Omron Sysmac Studio project CC087 Control System Demo 2.0 (Sysmac Studio 1.0.8.31, StandardProject)

# Controller new_Controller_0: NJ301-1100 version 1.6
Axis MC_Axis000, settings changed from default: AxisType=ServoType, HomingMode=LimitSignalOff, OriginInputMode=EXT, HomingVelocity=100000, HomingApproachVelocity=10000, OriginPositionOffset=1000
Task PrimaryTask (priority 4, period or condition 1000): Program0

VAR_GLOBAL
    CounterVariable1 : INT := 0;
    NB_Size AT %W3 : INT := 0;
    NB_Color AT %W4 : INT;
END_VAR
VAR_GLOBAL RETAIN
    ErrorMessage AT %H0.02 : BOOL;
END_VAR
VAR_GLOBAL
    NumberSelected : INT := 0;
    NB_A AT %W0.08 : BOOL;
    NB_B AT %W0.10 : BOOL;
    NB_C AT %W0.11 : BOOL;
    NB_D AT %W0.12 : BOOL;
    NB_E AT %W0.13 : BOOL;
    NB_F AT %W0.14 : BOOL;
    NB_G AT %W0.15 : BOOL;
END_VAR
VAR_GLOBAL RETAIN
    NB_Black AT %H0.01 : BOOL;
END_VAR
VAR_GLOBAL
    NB_Blue AT %W0.09 : BOOL;
    NB_Green AT %W0.07 : BOOL;
    NB_OutputWord AT %W2 : STRING[256];
    NB_Word AT %W1 : INT;
    NB_Run AT %W0.02 : BOOL;
    NB_Power AT %W0.03 : BOOL;
    CounterVariable2 : INT := 0;
    CounterVariable3 : INT := 0;
    Motor : BOOL;
    GreenStartButtonLight : BOOL;  (* at ECAT://node#[2,2]/Output Bit 16 bits/Output Bit 03 *)
    SwOne : BOOL;
    SwTwo : BOOL;
    SwThree : BOOL;
    SwFour : BOOL;
    OutOne : BOOL;  (* at ECAT://node#[2,2]/Output Bit 16 bits/Output Bit 04 *)
    OutTwo : BOOL;  (* at ECAT://node#[2,2]/Output Bit 16 bits/Output Bit 05 *)
    OutThree : BOOL;  (* at ECAT://node#[2,2]/Output Bit 16 bits/Output Bit 06 *)
    OutFour : BOOL;  (* at ECAT://node#[2,2]/Output Bit 16 bits/Output Bit 07 *)
    OutFive : BOOL;
    ReadyStatus : BOOL;  (* at ECAT://node#[2,1]/Input Bit 16 bits/Input Bit 01 *)
    FaultStatus : BOOL;  (* at ECAT://node#[2,1]/Input Bit 16 bits/Input Bit 02 *)
    RunStatus : BOOL;
    ConditionOne : BOOL;  (* at ECAT://node#[2,1]/Input Bit 16 bits/Input Bit 00 *)
    ConditionTwo : BOOL;  (* at ECAT://node#[2,1]/Input Bit 16 bits/Input Bit 03 *)
    ConditionThree : BOOL;
    ConditionFour : BOOL;
    ConditionFive : BOOL;
    StandByMode : BOOL;
    GreenStackLight : BOOL;  (* at ECAT://node#[2,2]/Output Bit 16 bits/Output Bit 00 *)
    RedStackLight : BOOL;  (* at ECAT://node#[2,2]/Output Bit 16 bits/Output Bit 02 *)
    YellowStackLight : BOOL;  (* at ECAT://node#[2,2]/Output Bit 16 bits/Output Bit 01 *)
    Output1 : BOOL;
END_VAR
VAR_GLOBAL CONSTANT
    MC_Axis000 : _sAXIS_REF;  (* at MC://_MC_AX[0] *)
END_VAR

PROGRAM Program0
VAR
    DelayTimer1 : TON;
    ET1 : TIME;
    OnTimer1 : TP;
    ET2 : TIME;
    DelayTimer2 : TON;
    OnTimer2 : TP;
    ET3 : TIME;
    ET4 : TIME;
    DelayTimer3 : TON;
    OnTimer3 : TP;
    ET5 : TIME;
    ET6 : TIME;
    Output1 : BOOL;
    ConditionFour : BOOL;
    ConditionFive : BOOL;
    OutFive : BOOL;
    FaultTimer : TON;
    ET7 : TIME;
    Power1 : MC_Power;
    Move1 : MC_MoveRelative;
    Reset1 : MC_Reset;
    TestFunction : FunctionBlock0;
    TestInput : BOOL;
    TestOutput : BOOL;
    Output : BOOL;
    Fault : BOOL;
    Home1 : MC_Home;
END_VAR
VAR_EXTERNAL
    FaultStatus : BOOL;
    RedStackLight : BOOL;
    ReadyStatus : BOOL;
    YellowStackLight : BOOL;
    GreenStackLight : BOOL;
    StandByMode : BOOL;
    SwFour : BOOL;
    SwOne : BOOL;
    SwTwo : BOOL;
    SwThree : BOOL;
    GreenStartButtonLight : BOOL;
    ConditionOne : BOOL;
    ConditionTwo : BOOL;
    ConditionThree : BOOL;
    CounterVariable1 : INT;
    CounterVariable2 : INT;
    CounterVariable3 : INT;
    OutOne : BOOL;
    OutTwo : BOOL;
    OutThree : BOOL;
    OutFour : BOOL;
    NB_Run : BOOL;
END_VAR
VAR_EXTERNAL CONSTANT
    MC_Axis000 : _sAXIS_REF;
END_VAR
VAR_EXTERNAL
    NB_Power : BOOL;
    Motor : BOOL;
    NB_A : BOOL;
    NB_Green : BOOL;
    NB_OutputWord : STRING[256];
    NB_B : BOOL;
    NB_C : BOOL;
    NB_D : BOOL;
    NB_E : BOOL;
    NB_F : BOOL;
    NB_G : BOOL;
    NB_Black : BOOL;
    NB_Blue : BOOL;
    NumberSelected : INT;
    ErrorMessage : BOOL;
    NB_Size : INT;
    NB_Word : INT;
    NB_Color : INT;
END_VAR

(* Section Section0: ladder, written here as Structured Text *)

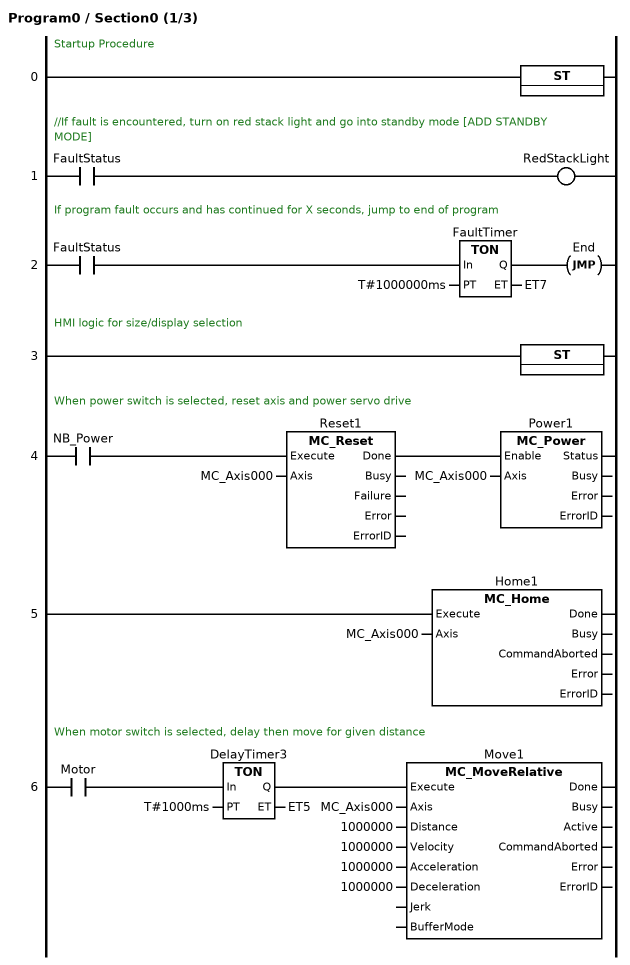
(* Rung 0: Startup Procedure *)
    
(* Rung 1: //If fault is encountered, turn on red stack light and go into standby mode [ADD STANDBY MODE] *)
RedStackLight := FaultStatus;
(* Rung 2: If program fault occurs and has continued for X seconds, jump to end of program *)
FaultTimer(In := FaultStatus, PT := T#1000000ms, ET => ET7);
IF FaultTimer.Q THEN JMP End; END_IF;
(* Rung 3: HMI logic for size/display selection *)
    
(* Rung 4: When power switch is selected, reset axis and power servo drive *)
Reset1(Execute := NB_Power, Axis := MC_Axis000);
Power1(Enable := Reset1.Done, Axis := MC_Axis000);
(* Rung 5 *)
Home1(Execute := TRUE, Axis := MC_Axis000);
(* Rung 6: When motor switch is selected, delay then move for given distance *)
DelayTimer3(In := Motor, PT := T#1000ms, ET => ET5);
Move1(Execute := DelayTimer3.Q, Axis := MC_Axis000, Distance := 1000000, Velocity := 1000000, Acceleration := 1000000, Deceleration := 1000000);

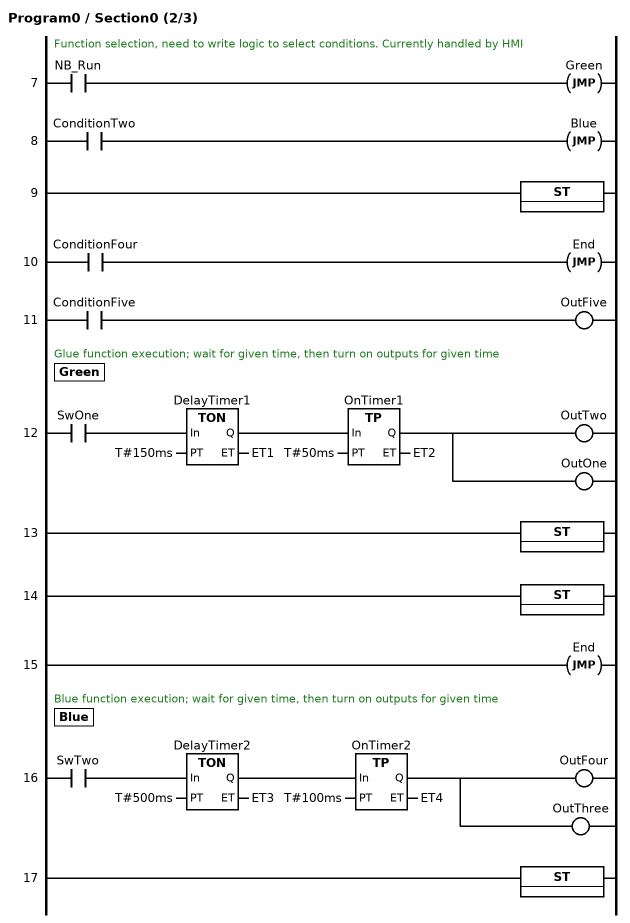
(* Rung 7: Function selection, need to write logic to select conditions. Currently handled by HMI *)
IF NB_Run THEN JMP Green; END_IF;
(* Rung 8 *)
IF ConditionTwo THEN JMP Blue; END_IF;
(* Rung 9 *)
    
(* Rung 10 *)
IF ConditionFour THEN JMP End; END_IF;
(* Rung 11 *)
OutFive := ConditionFive;
(* Rung 12: Glue function execution; wait for given time, then turn on outputs for given time *)
Green:
DelayTimer1(In := SwOne, PT := T#150ms, ET => ET1);
OnTimer1(In := DelayTimer1.Q, PT := T#50ms, ET => ET2);
OutTwo := OnTimer1.Q;
OutOne := OnTimer1.Q;
(* Rung 13 *)
    
(* Rung 14 *)
    
(* Rung 15 *)
JMP End;
(* Rung 16: Blue function execution; wait for given time, then turn on outputs for given time *)
Blue:
DelayTimer2(In := SwTwo, PT := T#500ms, ET => ET3);
OnTimer2(In := DelayTimer2.Q, PT := T#100ms, ET => ET4);
OutFour := OnTimer2.Q;
OutThree := OnTimer2.Q;
(* Rung 17 *)
    

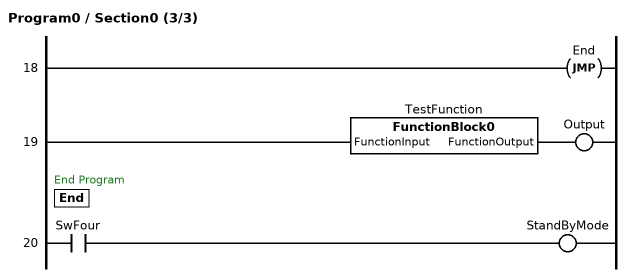
(* Rung 18 *)
JMP End;
(* Rung 19 *)
TestFunction(FunctionInput := TRUE);
Output := TestFunction.FunctionOutput;
(* Rung 20: End Program *)
End:
StandByMode := SwFour;
END_PROGRAM

FUNCTION_BLOCK FunctionBlock0
VAR
    TestInput : BOOL;
    Output : BOOL;
    Input : BOOL;
END_VAR
VAR_INPUT
    FunctionInput : BOOL;
END_VAR
VAR_OUTPUT
    FunctionOutput : BOOL;
END_VAR
VAR_EXTERNAL
    OutFive : BOOL;
END_VAR
(* ladder, written here as Structured Text *)

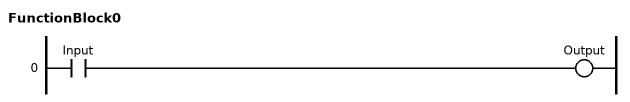
(* Rung 0 *)
Output := Input;
END_FUNCTION_BLOCK